// TIA Portal V19 export
DATA_BLOCK "Main_Safety_RTG1_DB"   // DB15, F_DB
NAME : FUSI
// stored: InstanceOfName Main_Safety_RTG1, InstanceOfType FB
"Main_Safety_RTG1"
BEGIN
END_DATA_BLOCK
